(* Logix 5000 project; controller CLASE_1 Emulate 5570 rev 28.11; software revision 28.02; part 2 of 15 *)
(* tags used below, declared in another part *)
   Inp_PVSrcQ : SINT;   // Input Source and Quality (from Channel object, if available) (enum)
   Inp_PVBad : BOOL;   // 1=PV or I/O Comms Status Bad, 0=OK
   Inp_PVUncertain : BOOL;   // 1=PV Value Not Reliable, 0=OK
   Inp_Sim : BOOL;   // 1=Use simulated PV (Set_SimPV); 0=Use Input (Inp_PV)
   Cfg_UseChanSrcQ : BOOL;   // 1=Pass thru connected Channel's SrcQ value, 0=generate SrcQ
   Cfg_HiHiDB : REAL;   // High-High Status Deadband (EU)
   Cfg_HiDB : REAL;   // High Status Deadband (EU)
   Cfg_LoDB : REAL;   // Low Status Deadband (EU)
   Cfg_LoLoDB : REAL;   // Low-Low Status Deadband (EU)
   Cfg_FailDB : REAL;   // Out-of-Range (fail) High/Low Deadband (EU)
   PSet_Owner : DINT;   // Program Owner Request ID (non-zero) or Release (zero)
   PCmd_ClearCapt : BOOL;   // Program Command to Clear the captured min / max PV excursion values
   MCmd_SubstPV : BOOL;   // Maintenance Command to use Substitute PV (override input)
   MCmd_InpPV : BOOL;   // Maintenance Command to use Input PV (normal)
   OCmd_ResetAckAll : BOOL;   // Operator Command to Reset and Acknowledge all Alarms
   Val : REAL;   // Analog Value (after Substitute PV, if used)
   Val_InpPV : REAL;   // Analog Input Value (actual, before Substitute PV selection)
   SrcQ_IO : SINT;   // Source and Quality of primary I/O (enumeration)
   SrcQ : SINT;   // Source and Quality of primary Val/Sts (enumeration)
   Val_Fault : SINT;   // Device Fault Status 0=none, 20=Lo, 21=Hi, 24=LoLo, 25=HiHi, 32=Fail, 34=CfgErr
   Val_Owner : DINT;   // Current Object Owner ID (0=not owned)
   Sts_SubstPV : BOOL;   // 1=Using Substitute PV (Input being overridden)
   Err_Raw : BOOL;   // 1=Error in Config: Raw Input Scaling Min = Max
   Err_EU : BOOL;   // 1=Error in Config: Scaled EU Min = Max
   Err_Filt : BOOL;   // 1=Error in Config: PV filter params (RateTime, TC)
   Err_DB : BOOL;   // 1=Error in Config: a Status Deadband is < 0.0
   Err_Alarm : BOOL;   // 1=Error in Config: Alarm Min On Time, Shelf Time, Severity
   Sts_HiHi : ALIAS FOR HiHi.Inp;   // 1=Analog Input is above High-High limit
   Sts_Hi : ALIAS FOR Hi.Inp;   // 1=Analog Input is above High limit
   Sts_Lo : ALIAS FOR Lo.Inp;   // 1=Analog Input is below Low limit
   Sts_LoLo : ALIAS FOR LoLo.Inp;   // 1=Analog Input is below Low-Low limit
   Sts_Fail : ALIAS FOR Fail.Inp;   // 1=Analog Input is Out of Range or PV Bad
   Rdy_ResetAckAll : BOOL;   // 1=At least one Alarm requires Reset or Acknowledgement
   P_AIn : BOOL;   // Unique Parameter Name for auto - discovery
   LoLo : P_Alarm;   // Low-Low Alarm
   Lo : P_Alarm;   // Low Alarm
   Hi : P_Alarm;   // High Alarm
   HiHi : P_Alarm;   // High-High Alarm
   Mode : P_Mode;   // Analog Input Mode Selection
   Fail : P_Alarm;   // Analog Input Failure Alarm (bad quality or out of range)
   Wrk_Notify : SINT;   // Buffer for building Val_Notify
   Wrk_Fault : SINT;   // Buffer for building Val_Fault
   Wrk_SrcQ : SINT;   // Register for building Source / Quality enumeration
   Wrk_ValidONS : BOOL;   // Selected PV goes from Infinite or Not a Number to VALID
   Wrk_SelPVInfNaN : BOOL;   // Selected PV (Input or Substitute) is Infinite or NaN
   FailGate : P_Gate;   // Fail Alarm Gate / Delay Block
   Wrk_InpInfNaN : BOOL;   // Input is Infinite or Not a Number
   Wrk_InpFail : BOOL;   // Input Fail: out of range
(* P_AIn, continued *)

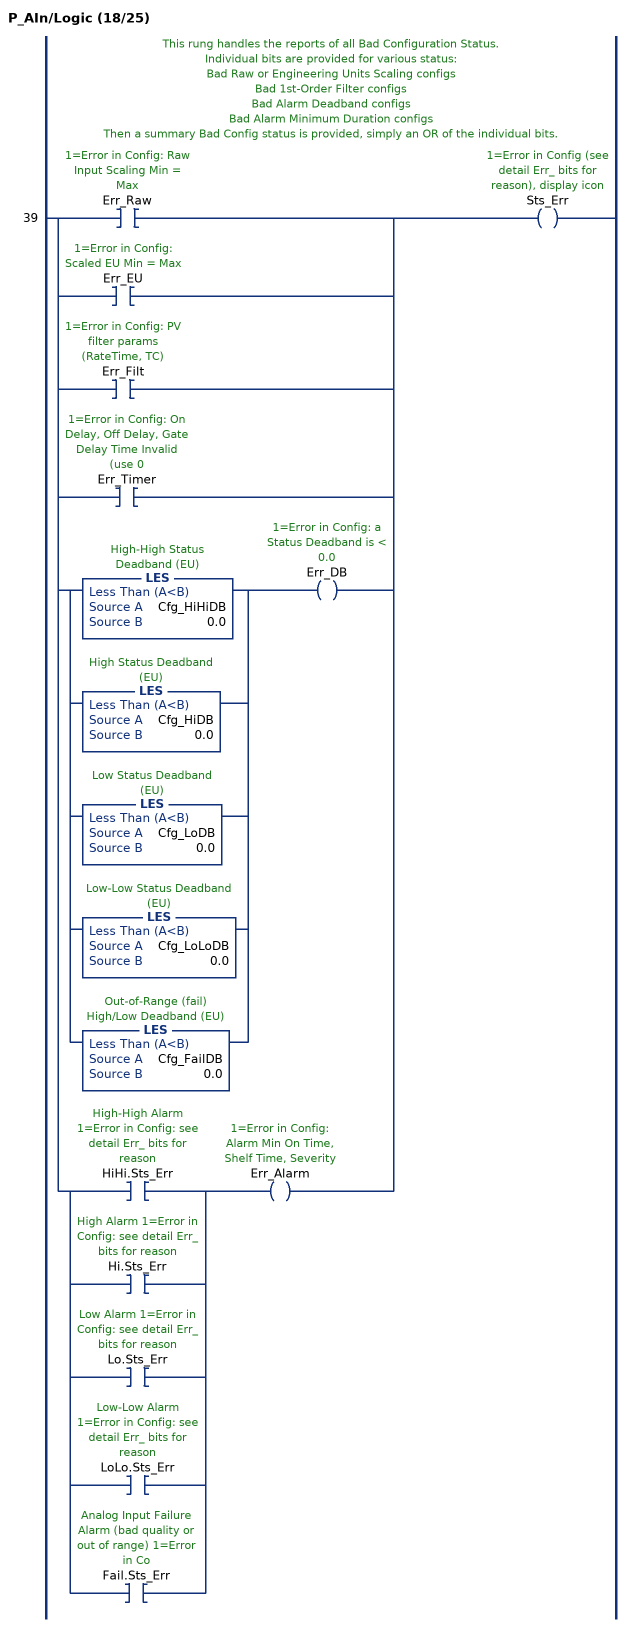
   // This rung handles the reports of all Bad Configuration Status.
   // Individual bits are provided for various status:
   // Bad Raw or Engineering Units Scaling configs
   // Bad 1st-Order Filter configs
   // Bad Alarm Deadband configs
   // Bad Alarm Minimum Duration configs
   // Then a summary Bad Config status is provided, simply an OR of the individual bits.
   39: [XIC(Err_Raw) ,XIC(Err_EU) ,XIC(Err_Filt) ,XIC(Err_Timer) ,[LES(Cfg_HiHiDB,0.0) ,LES(Cfg_HiDB,0.0) ,LES(Cfg_LoDB,0.0) ,LES(Cfg_LoLoDB,0.0) ,LES(Cfg_FailDB,0.0) ] OTE(Err_DB) ,[XIC(HiHi.Sts_Err) ,XIC(Hi.Sts_Err) ,XIC(Lo.Sts_Err) ,XIC(LoLo.Sts_Err) ,XIC(Fail.Sts_Err) ] OTE(Err_Alarm) ]OTE(Sts_Err);
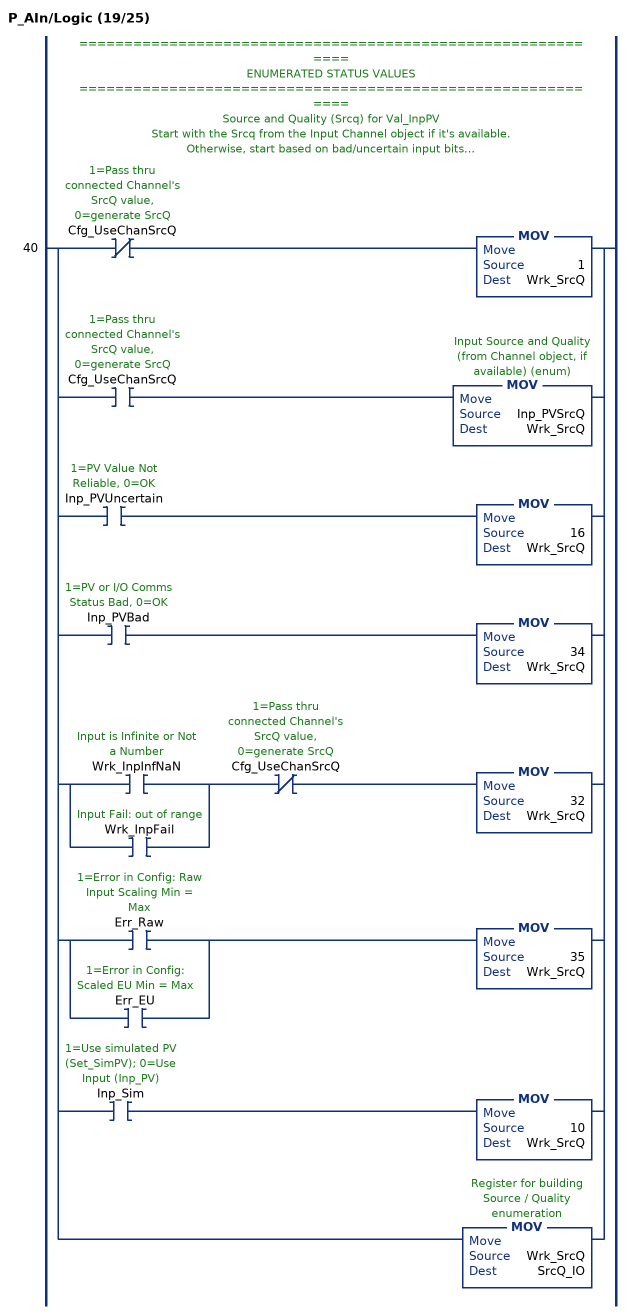
   // ============================================================
   // ENUMERATED STATUS VALUES
   // ============================================================
   // Source and Quality (Srcq) for Val_InpPV
   // Start with the Srcq from the Input Channel object if it's available.
   // Otherwise, start based on bad/uncertain input bits.
   // 0 = Good: live, confirmed good;   1 = Good: live, assumed good;
   // 2 = Good: no feedback, assumed good;   8 = Test: Simulated;   9 = Test: Loopback;
   // 10 = Test: Manually Entered;   16 = Uncertain: Live, off-spec;
   // 17 = Uncertain, Substituted at Device / Bus;   18 = Uncertain, Substituted at AOI;
   // 19 = Uncertain, using last known good;    20 = Uncertain, using replacement value;
   // 32 = Bad, Signal Failure;   33 = Bad, Channel Fault;
   // 34 = Bad, Module / Comms Fault;   35 = Bad, Invalid Configuration
   // #####  V3.1-00  2014-06-30:  Added rung for Source/Quality enumerations.  #####
   // #####  V3.5-02  2016-03-28:  Modified to add Cfg_UseChanSrcQ.  #####
   40: [XIO(Cfg_UseChanSrcQ) MOV(1,Wrk_SrcQ) ,XIC(Cfg_UseChanSrcQ) MOV(Inp_PVSrcQ,Wrk_SrcQ) ,XIC(Inp_PVUncertain) MOV(16,Wrk_SrcQ) ,XIC(Inp_PVBad) MOV(34,Wrk_SrcQ) ,[XIC(Wrk_InpInfNaN) ,XIC(Wrk_InpFail) ] XIO(Cfg_UseChanSrcQ) MOV(32,Wrk_SrcQ) ,[XIC(Err_Raw) ,XIC(Err_EU) ] MOV(35,Wrk_SrcQ) ,XIC(Inp_Sim) MOV(10,Wrk_SrcQ) ,MOV(Wrk_SrcQ,SrcQ_IO) ];
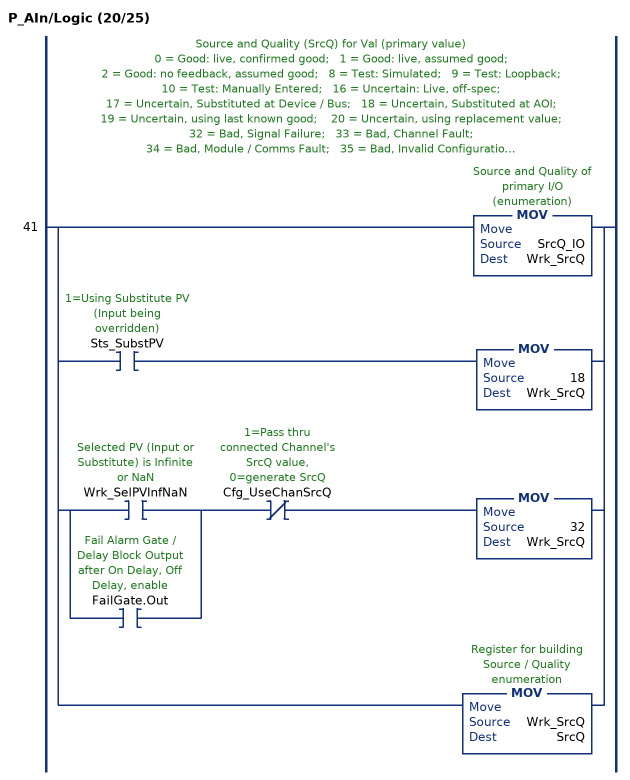
   // Source and Quality (SrcQ) for Val (primary value)
   // 0 = Good: live, confirmed good;   1 = Good: live, assumed good;
   // 2 = Good: no feedback, assumed good;   8 = Test: Simulated;   9 = Test: Loopback;
   // 10 = Test: Manually Entered;   16 = Uncertain: Live, off-spec;
   // 17 = Uncertain, Substituted at Device / Bus;   18 = Uncertain, Substituted at AOI;
   // 19 = Uncertain, using last known good;    20 = Uncertain, using replacement value;
   // 32 = Bad, Signal Failure;   33 = Bad, Channel Fault;
   // 34 = Bad, Module / Comms Fault;   35 = Bad, Invalid Configuration
   // #####  V3.1-00  2014-06-30:  Added rung for Source/Quality enumerations.  #####
   // #####  V3.5-02  2016-03-28:  Modified to add Cfg_UseChanSrcQ.  #####
   41: [MOV(SrcQ_IO,Wrk_SrcQ) ,XIC(Sts_SubstPV) MOV(18,Wrk_SrcQ) ,[XIC(Wrk_SelPVInfNaN) ,XIC(FailGate.Out) ] XIO(Cfg_UseChanSrcQ) MOV(32,Wrk_SrcQ) ,MOV(Wrk_SrcQ,SrcQ) ];
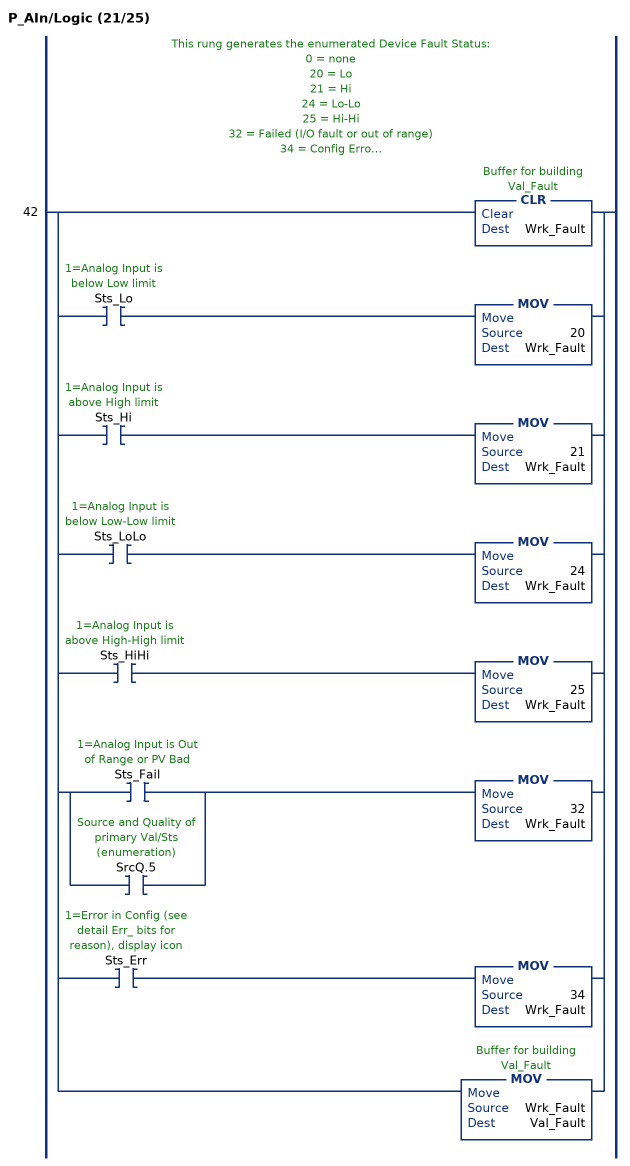
   // This rung generates the enumerated Device Fault Status:
   // 0 = none
   // 20 = Lo
   // 21 = Hi
   // 24 = Lo-Lo
   // 25 = Hi-Hi
   // 32 = Failed (I/O fault or out of range)
   // 34 = Config Error
   // #####  V3.1-05  2016-01-22:  Added check of SrcQ >= 32 for Val_Fault.  #####
   42: [CLR(Wrk_Fault) ,XIC(Sts_Lo) MOV(20,Wrk_Fault) ,XIC(Sts_Hi) MOV(21,Wrk_Fault) ,XIC(Sts_LoLo) MOV(24,Wrk_Fault) ,XIC(Sts_HiHi) MOV(25,Wrk_Fault) ,[XIC(Sts_Fail) ,XIC(SrcQ.5) ] MOV(32,Wrk_Fault) ,XIC(Sts_Err) MOV(34,Wrk_Fault) ,MOV(Wrk_Fault,Val_Fault) ];
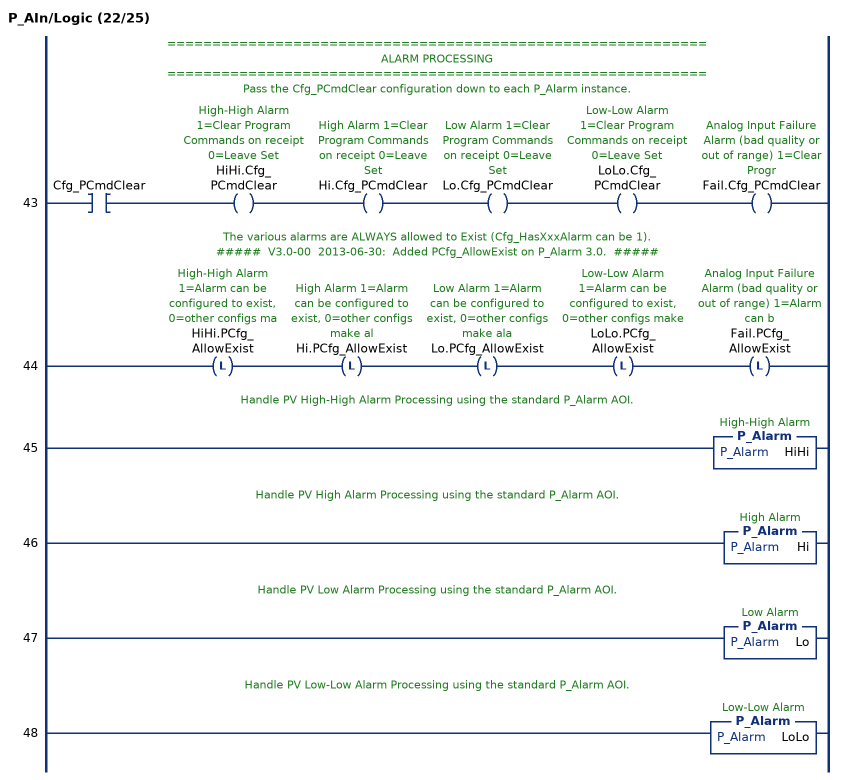
   // ============================================================
   // ALARM PROCESSING
   // ============================================================
   // Pass the Cfg_PCmdClear configuration down to each P_Alarm instance.
   43: XIC(Cfg_PCmdClear)OTE(HiHi.Cfg_PCmdClear)OTE(Hi.Cfg_PCmdClear)OTE(Lo.Cfg_PCmdClear)OTE(LoLo.Cfg_PCmdClear)OTE(Fail.Cfg_PCmdClear);
   // The various alarms are ALWAYS allowed to Exist (Cfg_HasXxxAlarm can be 1).
   // #####  V3.0-00  2013-06-30:  Added PCfg_AllowExist on P_Alarm 3.0.  #####
   44: OTL(HiHi.PCfg_AllowExist)OTL(Hi.PCfg_AllowExist)OTL(Lo.PCfg_AllowExist)OTL(LoLo.PCfg_AllowExist)OTL(Fail.PCfg_AllowExist);
   // Handle PV High-High Alarm Processing using the standard P_Alarm AOI.
   45: P_Alarm(HiHi);
   // Handle PV High Alarm Processing using the standard P_Alarm AOI.
   46: P_Alarm(Hi);
   // Handle PV Low Alarm Processing using the standard P_Alarm AOI.
   47: P_Alarm(Lo);
   // Handle PV Low-Low Alarm Processing using the standard P_Alarm AOI.
   48: P_Alarm(LoLo);
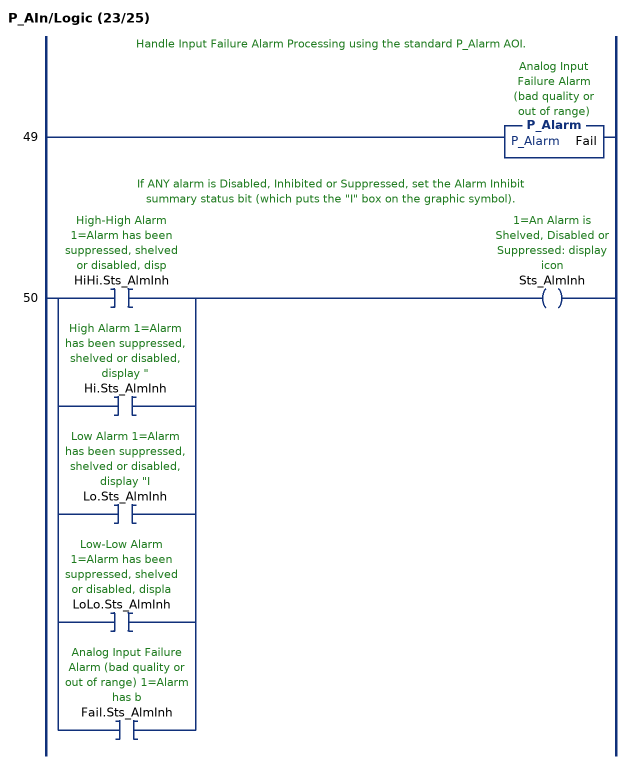
   // Handle Input Failure Alarm Processing using the standard P_Alarm AOI.
   49: P_Alarm(Fail);
   // If ANY alarm is Disabled, Inhibited or Suppressed, set the Alarm Inhibit
   // summary status bit (which puts the "I" box on the graphic symbol).
   50: [XIC(HiHi.Sts_AlmInh) ,XIC(Hi.Sts_AlmInh) ,XIC(Lo.Sts_AlmInh) ,XIC(LoLo.Sts_AlmInh) ,XIC(Fail.Sts_AlmInh) ]OTE(Sts_AlmInh);
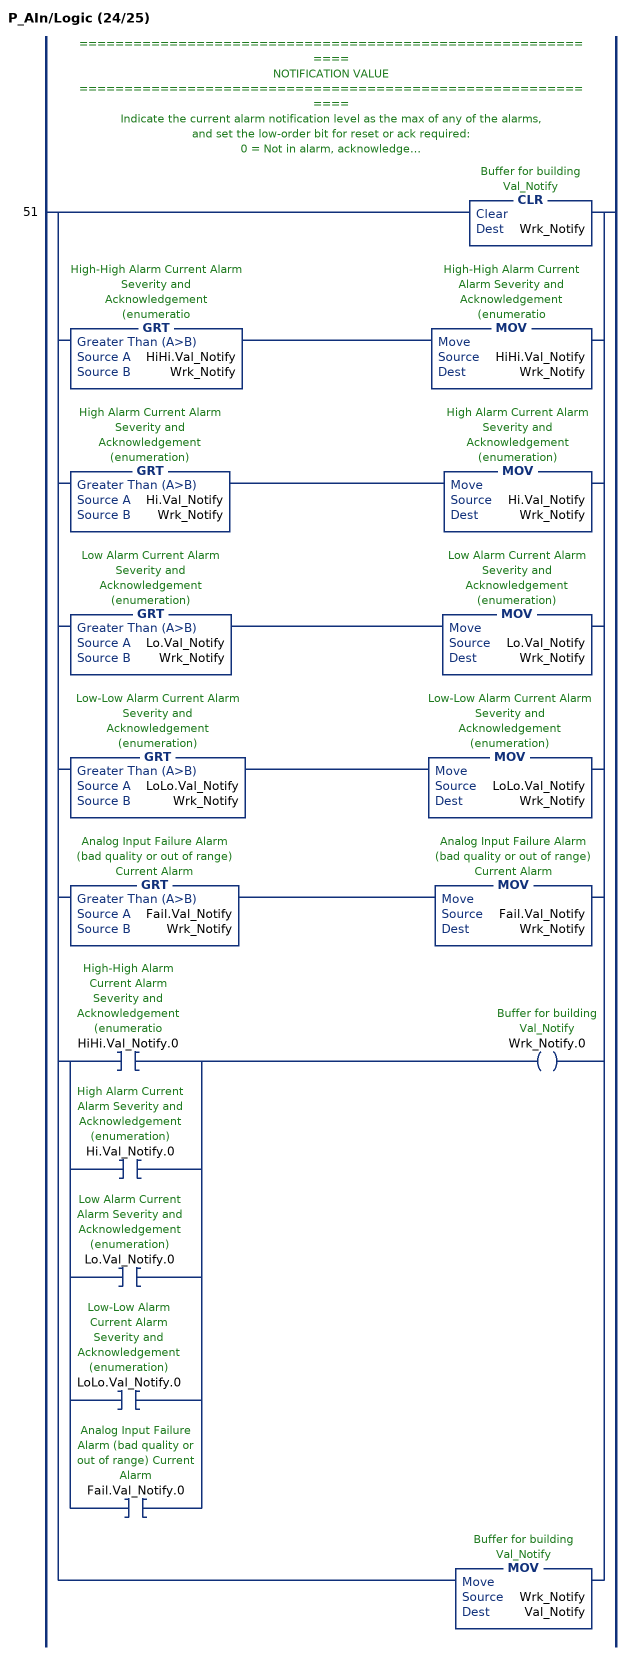
   // ============================================================
   // NOTIFICATION VALUE
   // ============================================================
   // Indicate the current alarm notification level as the max of any of the alarms,
   // and set the low-order bit for reset or ack required:
   // 0 = Not in alarm, acknowledged
   // 1 = Not in alarm, unacknowledged or reset required
   // 2 = Low severity alarm, acknowledged
   // 3 = Low severity alarm, unacknowledged
   // 4 = Medium severity alarm, acknowledged
   // 5 = Medium severity alarm, unacknowledged
   // 6 = High severity alarm, acknowledged
   // 7 = High severity alarm, unacknowledged
   // 8 = Urgent severity alarm, acknowledged
   // 9 = Urgent severity alarm, unacknowledged
   // #####  V3.1-00  2014-06-30:  Separated Reset Reqd functions from Val_Notify  #####
   51: [CLR(Wrk_Notify) ,GRT(HiHi.Val_Notify,Wrk_Notify) MOV(HiHi.Val_Notify,Wrk_Notify) ,GRT(Hi.Val_Notify,Wrk_Notify) MOV(Hi.Val_Notify,Wrk_Notify) ,GRT(Lo.Val_Notify,Wrk_Notify) MOV(Lo.Val_Notify,Wrk_Notify) ,GRT(LoLo.Val_Notify,Wrk_Notify) MOV(LoLo.Val_Notify,Wrk_Notify) ,GRT(Fail.Val_Notify,Wrk_Notify) MOV(Fail.Val_Notify,Wrk_Notify) ,[XIC(HiHi.Val_Notify.0) ,XIC(Hi.Val_Notify.0) ,XIC(Lo.Val_Notify.0) ,XIC(LoLo.Val_Notify.0) ,XIC(Fail.Val_Notify.0) ] OTE(Wrk_Notify.0) ,MOV(Wrk_Notify,Val_Notify) ];
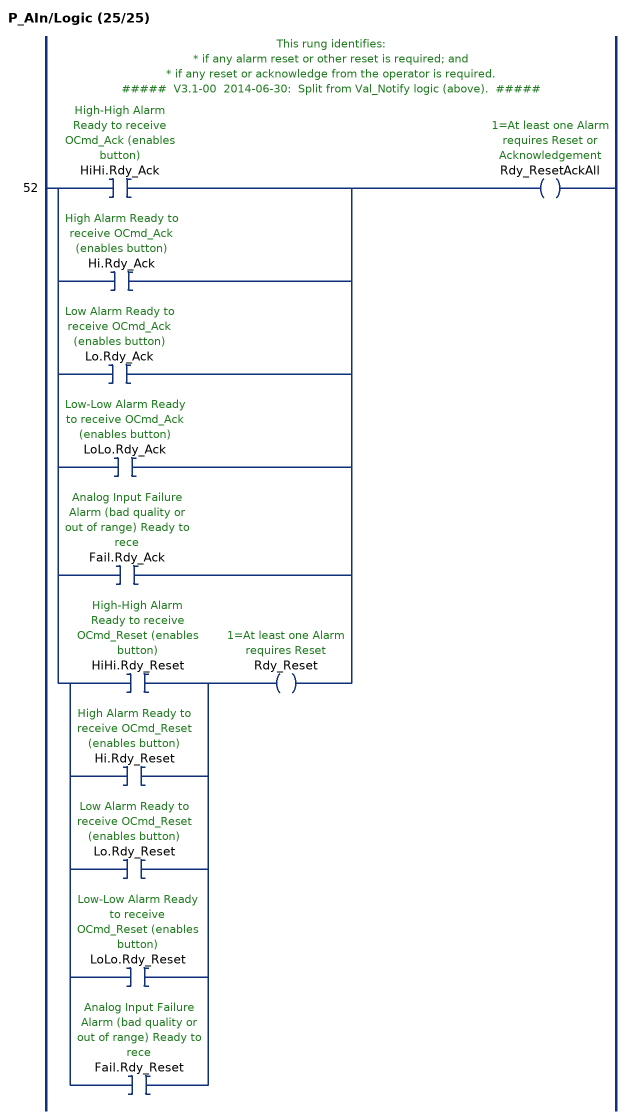
   // This rung identifies:
   // * if any alarm reset or other reset is required; and
   // * if any reset or acknowledge from the operator is required.
   // #####  V3.1-00  2014-06-30:  Split from Val_Notify logic (above).  #####
   52: [[XIC(HiHi.Rdy_Ack) ,XIC(Hi.Rdy_Ack) ,XIC(Lo.Rdy_Ack) ,XIC(LoLo.Rdy_Ack) ,XIC(Fail.Rdy_Ack) ] ,[XIC(HiHi.Rdy_Reset) ,XIC(Hi.Rdy_Reset) ,XIC(Lo.Rdy_Reset) ,XIC(LoLo.Rdy_Reset) ,XIC(Fail.Rdy_Reset) ] OTE(Rdy_Reset) ]OTE(Rdy_ResetAckAll);
END_ROUTINE

ROUTINE Prescan   (* ladder *)
// Clear Ownership. clear "lurking" Commands
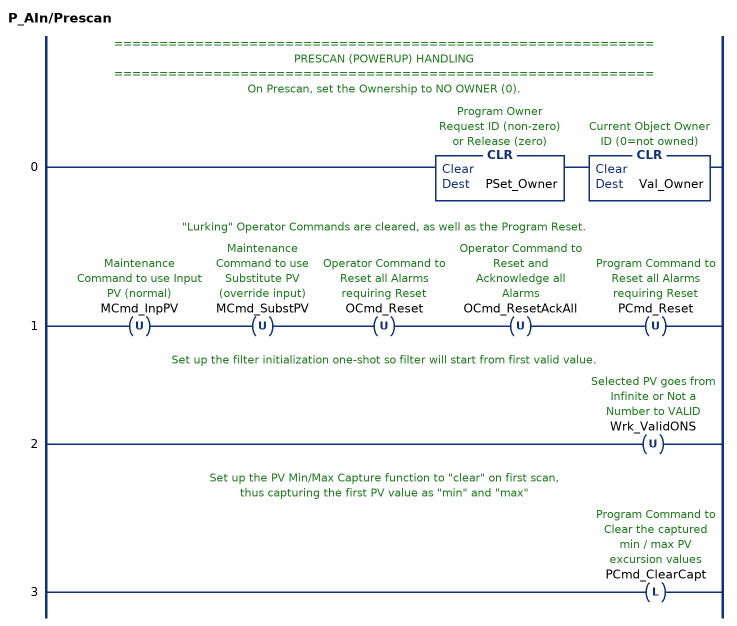
   // ============================================================
   // PRESCAN (POWERUP) HANDLING
   // ============================================================
   // On Prescan, set the Ownership to NO OWNER (0).
   0: CLR(PSet_Owner)CLR(Val_Owner);
   // "Lurking" Operator Commands are cleared, as well as the Program Reset.
   1: OTU(MCmd_InpPV)OTU(MCmd_SubstPV)OTU(OCmd_Reset)OTU(OCmd_ResetAckAll)OTU(PCmd_Reset);
   // Set up the filter initialization one-shot so filter will start from first valid value.
   2: OTU(Wrk_ValidONS);
   // Set up the PV Min/Max Capture function to "clear" on first scan,
   // thus capturing the first PV value as "min" and "max"
   3: OTL(PCmd_ClearCapt);
END_ROUTINE
END_ADD_ON_INSTRUCTION

ADD_ON_INSTRUCTION P_Alarm   (* revision 3.5 07Patch01 Release, vendor Rockwell Automation, ExecutePrescan, ExecuteEnableInFalse *)
// Alarm
// Revision note:
// See V3.5-xx Release Notes for details. Modified for FTView ME "chattering alarm" acknowledge timing.
// Help:
// Copyright © Rockwell Automation, Inc.  All Rights Reserved.
// This instruction monitors one input condition and provides one Alarm with:
//   * configurable latching (reset required) and acknowledgement requirement
//   * configurable alarm severity
//       1 to 250       = Low  (blue, typ. informational)
//       251 to 500   = Medium  (yelllow, typ. warning)
//       501 to 750   = High  (red, typ. process exception)
//       751 to 1000 = Urgent  (magenta, typ. equip. fault)
//   * configurable minimum ON time (e.g., to ensure it is seen by the HMI)
//   * commands to suppress/unsuppress (Prog), shelve/unshelve (Oper)
//         and disable/enable (Maint) the alarm.
//   * configurable amount of time shelved to automatically unshelve an alarm
//   * FTA&E support for suppressed, shelved and disabled states (V7.0)
//   * A Maintenance "Test" command, which triggers the alarm for the minimum
//      alarm time for testing purposes.
// NOTE regarding parameter naming:
//   FTAE names (same as ALMD instruction) are used instead
//   of the ANSI/ISA 18.2-2009 names, as follows:
//    "Disabled" is the equivalent of "Out of Service" in ISA 18.2.
//       (The Disabled state is owned by Maintenance.)
//    "Suppressed" is the equivalent of "Suppressed by Design" in
//       ISA 18.2. (The Suppressed state is owned by Program logic.)
//    "Shelved" is the same as in ISA 18.2.
//       (The Shelved state is owned by Operator, but may be cleared
//       by Program logic based on time, shift change, etc.)
// This instruction is usually nested within other instructions, with one instance
// used for each Alarm generated by the containing instruction.  It may also be
// used as a standalone instruction for Alarm conditions generated by custom logic.
// FTAE Alarm Setup:
//   (object).(alarm).Com_AE.0:  Alarm to FTAE
//     .Com_AE.1:   Ack to/from FTAE
//     .Com_AE.3:   Shelved from FTAE Status
//     .Com_AE.4:   Shelve/Reshelve to FTAE Control (auto reset)
//     .Com_AE.5:   Unshelve to FTAE Control (auto reset)
//     .Com_AE.6:   Suppressed from FTAE Status
//     .Com_AE.7:   Suppress to FTAE Control (auto reset)
//     .Com_AE.8:   Unsuppress to FTAE Control (auto reset)
//     .Com_AE.9:   Disabled from FTAE Status
//     .Com_AE.10: Disable to FTAE Control (auto reset)
//     .Com_AE.11: Enable to FTAE Control (auto reset)
//    all other bits unused
//     .Cfg_MaxShelfT is also used in FTAE config.
//     .Cfg_Severity is used in FTAE for FTView 8.x.
VAR_INPUT
   Inp : BOOL := 1; {visible}   // Alarm Condition Input 1=Alarm
   Inp_Reset : BOOL; {visible}   // 1=Reset Alarm requiring reset
   Cfg_Exists : BOOL := 1;   // 1=Alarm configured to exist, 0=Does not exist, don't scan
   Cfg_ResetReqd : BOOL;   // 1=Latched Alarm, a Reset is required to clear this Alarm
   Cfg_AckReqd : BOOL := 1;   // 1=Acknowledge required for this Alarm
   Cfg_AllowShelve : BOOL := 1;   // 1=Allow Operator to Shelve this Alarm
   Cfg_AllowDisable : BOOL := 1;   // 1=Allow Maintenance to Disable this Alarm
   Cfg_PCmdClear : BOOL := 1;   // 1=Clear Program Commands on receipt 0=Leave Set
   Cfg_Severity : INT := 750;   // Alarm Severity: 1..250=Low, 251..500=Medium, 501..750=High, 751..1000=Urgent
   Cfg_AlmMinOnT : DINT := 5;   // Minimum time Alm output stays on (sec)
   Cfg_MaxShelfT : INT := 480;   // Auto unshelve after shelved this long (1..32767 minutes)
   PCfg_AllowExist : BOOL := 1;   // 1=Alarm can be configured to exist, 0=other configs make alarm meaningless
   PCmd_Reset : BOOL;   // Program Command to Reset latched alarm
   PCmd_Ack : BOOL;   // Program Command to Acknowledge alarm
   PCmd_Suppress : BOOL;   // Program Command to Suppress by Design (inhibits new alarm)
   PCmd_Unsuppress : BOOL;   // Program Command to Unsuppress (allows new alarm)
   PCmd_Unshelve : BOOL;   // Program Command to Unshelve (e.g., on shift change)
   OCmd_Reset : BOOL;   // Operator Command to Reset latched alarm
   OCmd_Ack : BOOL;   // Operator Command to Acknowledge alarm
   OCmd_Shelve : BOOL;   // Operator Command to Shelve Alarm (inhibits new alarm)
   OCmd_Unshelve : BOOL;   // Operator Command to Unshelve alarm (allows new alarm)
   MCmd_Disable : BOOL;   // Maintenance Command to Disable alarm (inhibits new alarm)
   MCmd_Enable : BOOL;   // Maintenance Command to Enable alarm (allows new alarm)
   MCmd_Test : BOOL;   // Maintenance Command to Test alarm (issued for minimum alarm time)
END_VAR
VAR_OUTPUT
   Val_Notify : SINT; {access Read Only}   // Current Alarm Severity and Acknowledgement (enumeration)
   Val_MinToUnshelve : DINT; {access Read Only, visible}   // Number of minutes until this alarm unshelves itself (mmm:ss)
   Val_SecToUnshelve : DINT; {access Read Only, visible}   // Number of Seconds until this alarm unshelves itself (mmm:ss)
   Alm : ALIAS FOR Com_AE.0; {visible}   // Alarm output 1=In Alarm
   Ack : ALIAS FOR Com_AE.1; {visible}   // Alarm acknowledged status: 1=Ack rcvd
   Shelved : ALIAS FOR Com_AE.3; {visible}   // 1=Alarm has been Shelved by Operator (inhibits new alarm)
   Suppressed : ALIAS FOR Com_AE.6; {visible}   // 1=Alarm has been Suppressed by Program (inhibits new alarm)
   Disabled : ALIAS FOR Com_AE.9; {visible}   // 1=Alarm has been Disabled by Maintanance (inhibits new alarm)
   Sts_AlmInh : BOOL; {access Read Only}   // 1=Alarm has been suppressed, shelved or disabled, display "I" icon
   Sts_Err : BOOL; {access Read Only}   // 1=Error in Config: see detail Err_ bits for reason
   Err_Timer : BOOL; {access Read Only}   // 1=Error in Config: Alarm Min On Time, Shelf Time (use 0 to 2147483)
   Err_Severity : BOOL; {access Read Only}   // 1=Error in Config: Invalid Severity (use 1 to 4)
   Rdy_Reset : BOOL; {access Read Only}   // Ready to receive OCmd_Reset (enables button)
   Rdy_Ack : BOOL; {access Read Only}   // Ready to receive OCmd_Ack (enables button)
   Rdy_Shelve : BOOL; {access Read Only}   // Ready to receive OCmd_Shelve (enables button)
   Rdy_Unshelve : BOOL; {access Read Only}   // Ready to receive OCmd_Unshelve (enables button)
   Rdy_Disable : BOOL; {access Read Only}   // Ready to receive MCmd_Disable (enables button)
   Rdy_Enable : BOOL; {access Read Only}   // Ready to receive MCmd_Enable (enables button)
   Rdy_Test : BOOL; {access Read Only}   // Ready to receive MCmd_Test (enables button)
   P_Alarm : BOOL;   // Unique Parameter Name for auto - discovery
END_VAR
VAR
   Wrk_Alm : BOOL; {access None}   // Internal Alarm Status
   Wrk_Suppressed : BOOL; {access None}   // Internal Alarm Suppressed Status
   Wrk_AlmMinOnT : TIMER := (PRE := 5000); {access None}   // Alarm output minimum ON time to be seen by alarm server
   Wrk_AutoAckT : TIMER := (PRE := 5000); {access None}   // Time to clear Ack bit when Ack not required
   Wrk_ShelfT : TIMER; {access Read Only}   // Time to auto Unshelve a Shelved Alarm
   Inf_Tab : SINT;   // Tab to display (FTView ME)
   Com_AE : INT := 2#0000_0000_0000_0010;   // Communication with HMI / Alarm/Event Server (see bit descriptions)
        .0   // Alarm to AE
        .1   // Acked from AE Status, Ack to AE Control
        .10   // Disable to AE Control
        .11   // Enable to AE Control
        .12   // (not used)
        .13   // (not used)
        .14   // (not used)
        .15   // (not used)
        .2   // (not used)
        .3   // Shelved from AE Status
        .4   // Shelve to AE Control
        .5   // Unshelve to AE Control
        .6   // Suppressed from AE Status
        .7   // Suppress to AE Control
        .8   // Unsuppress to AE Control
        .9   // Disabled from AE Status
   Cfg_Tag : STRING_20 := 'P_Alarm';   // Alarm Tag Text (e.g., "LAHH-101")
   Cfg_Cond : STRING_20 := 'Alarm Condition';   // Alarm Condition Text (e.g., "High-High PV")
   Wrk_SecToUnshelve : DINT; {access None}   // Number of seconds until this alarm unshelves itself
   Inf_Lib : STRING_12 := 'RA-BAS'; {access Read Only}   // Display Library for Faceplate call-up
   Inf_Type : STRING_16 := 'P_Alarm'; {access Read Only}   // Must contain AOI name, used for HMI and Information S/W
END_VAR

ROUTINE EnableInFalse   (* ladder *)
// Perform Alarm processing, but Invert Alarm Input ("Inp") for use on LD rung (EnableIn False)
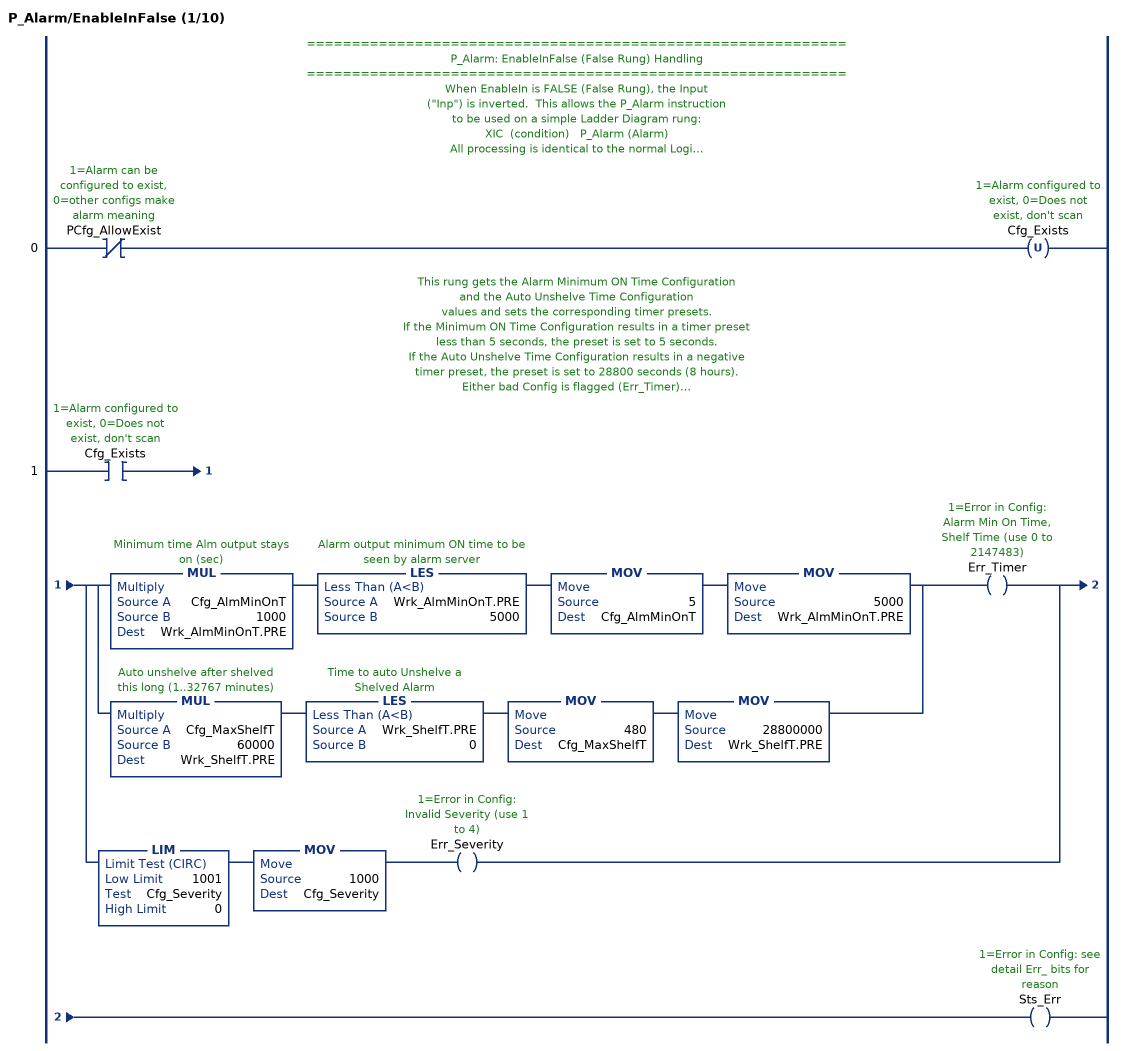
   // ============================================================
   // P_Alarm: EnableInFalse (False Rung) Handling
   // ============================================================
   // When EnableIn is FALSE (False Rung), the Input
   // ("Inp") is inverted.  This allows the P_Alarm instruction
   // to be used on a simple Ladder Diagram rung:
   // XIC  (condition)   P_Alarm (Alarm)
   // All processing is identical to the normal Logic
   // routine, except references to Inp are inverted!
   // ============================================================
   // CONFIGURATION
   // ============================================================
   // In the object containing this alarm, other configuration (such as not having
   // any limit switches) may make this particular alarm meaningless.
   // The Program Configuration "Allow Exist" is used to hide this alarm
   // on the object's faceplate and other graphics, and forces the Cfg_Exist to 0.
   // #####  V3.0-00  2013-06-30:  Added PCfg_AllowExist.  #####
   0: XIO(PCfg_AllowExist)OTU(Cfg_Exists);
   // This rung gets the Alarm Minimum ON Time Configuration
   // and the Auto Unshelve Time Configuration
   // values and sets the corresponding timer presets.
   // If the Minimum ON Time Configuration results in a timer preset
   // less than 5 seconds, the preset is set to 5 seconds.
   // If the Auto Unshelve Time Configuration results in a negative
   // timer preset, the preset is set to 28800 seconds (8 hours).
   // Either bad Config is flagged (Err_Timer).
   // Bad Config is also flagged if the Cfg_Severity is out of range (valid = 1..1000) (Err_Severity).
   // #####  V3.0-00  2013-06-30:  Changed Program Inhibit to Suppress, Operator Suppress to Shelve.  #####
   // #####  Added Shelf Timer config check; if Severity out of range, make it "Fault".  #####
   // #####  V3.0-02  2013-10-30:  Changed Cfg_MaxShelfT check to LEQ 0.  (INT 1 to 32767 is valid.)  #####
   // #####  V3.1-05, V3.5-00  2015-07-31:  Fixed operation of Cfg_MaxShelfT = 0, Cfg_AlmMinOnT, rung comment.  #####
   1: XIC(Cfg_Exists)[[MUL(Cfg_AlmMinOnT,1000,Wrk_AlmMinOnT.PRE) LES(Wrk_AlmMinOnT.PRE,5000) MOV(5,Cfg_AlmMinOnT) MOV(5000,Wrk_AlmMinOnT.PRE) ,MUL(Cfg_MaxShelfT,60000,Wrk_ShelfT.PRE) LES(Wrk_ShelfT.PRE,0) MOV(480,Cfg_MaxShelfT) MOV(28800000,Wrk_ShelfT.PRE) ] OTE(Err_Timer) ,LIM(1001,Cfg_Severity,0) MOV(1000,Cfg_Severity) OTE(Err_Severity) ]OTE(Sts_Err);
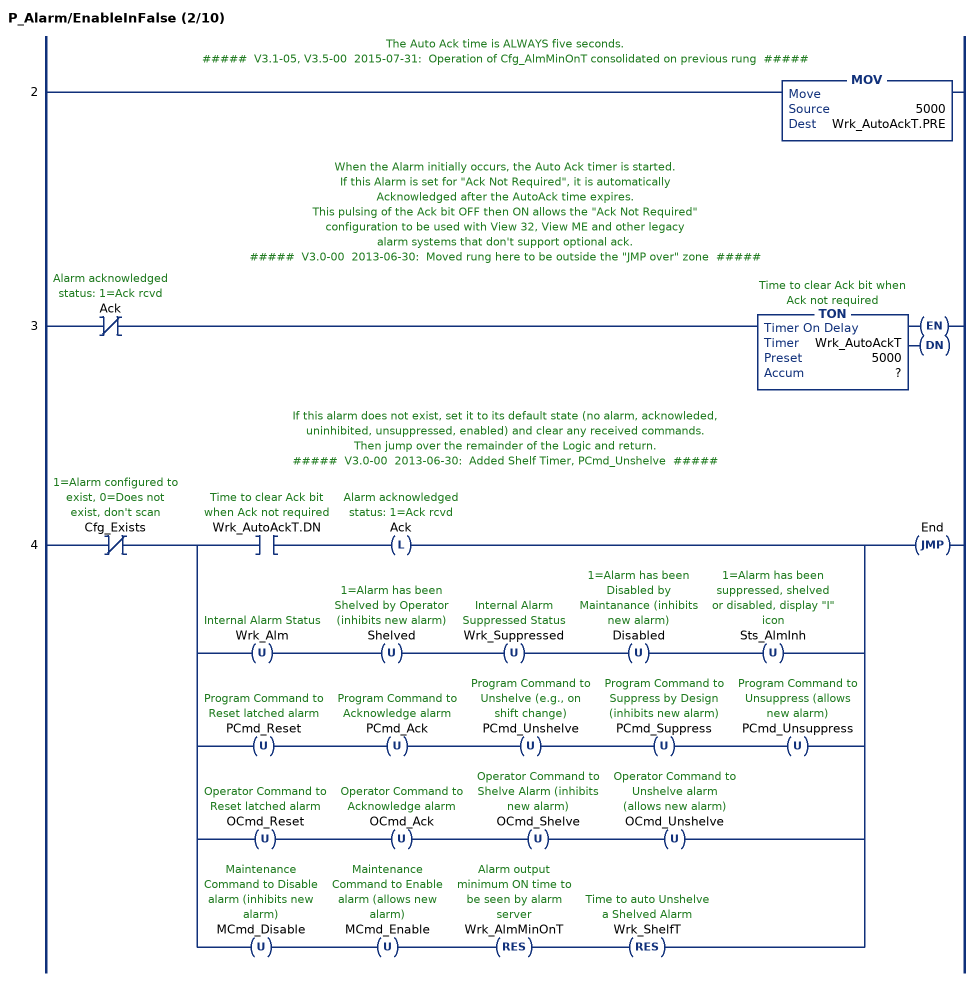
   // The Auto Ack time is ALWAYS five seconds.
   // #####  V3.1-05, V3.5-00  2015-07-31:  Operation of Cfg_AlmMinOnT consolidated on previous rung  #####
   2: MOV(5000,Wrk_AutoAckT.PRE);
   // When the Alarm initially occurs, the Auto Ack timer is started.
   // If this Alarm is set for "Ack Not Required", it is automatically
   // Acknowledged after the AutoAck time expires.
   // This pulsing of the Ack bit OFF then ON allows the "Ack Not Required"
   // configuration to be used with View 32, View ME and other legacy
   // alarm systems that don't support optional ack.
   // #####  V3.0-00  2013-06-30:  Moved rung here to be outside the "JMP over" zone  #####
   3: XIO(Ack)TON(Wrk_AutoAckT,?,?);
   // If this alarm does not exist, set it to its default state (no alarm, acknowleded,
   // uninhibited, unsuppressed, enabled) and clear any received commands.
   // Then jump over the remainder of the Logic and return.
   // #####  V3.0-00  2013-06-30:  Added Shelf Timer, PCmd_Unshelve  #####
   4: XIO(Cfg_Exists)[XIC(Wrk_AutoAckT.DN) OTL(Ack) ,OTU(Wrk_Alm) OTU(Shelved) OTU(Wrk_Suppressed) OTU(Disabled) OTU(Sts_AlmInh) ,OTU(PCmd_Reset) OTU(PCmd_Ack) OTU(PCmd_Unshelve) OTU(PCmd_Suppress) OTU(PCmd_Unsuppress) ,OTU(OCmd_Reset) OTU(OCmd_Ack) OTU(OCmd_Shelve) OTU(OCmd_Unshelve) ,OTU(MCmd_Disable) OTU(MCmd_Enable) RES(Wrk_AlmMinOnT) RES(Wrk_ShelfT) ]JMP(End);
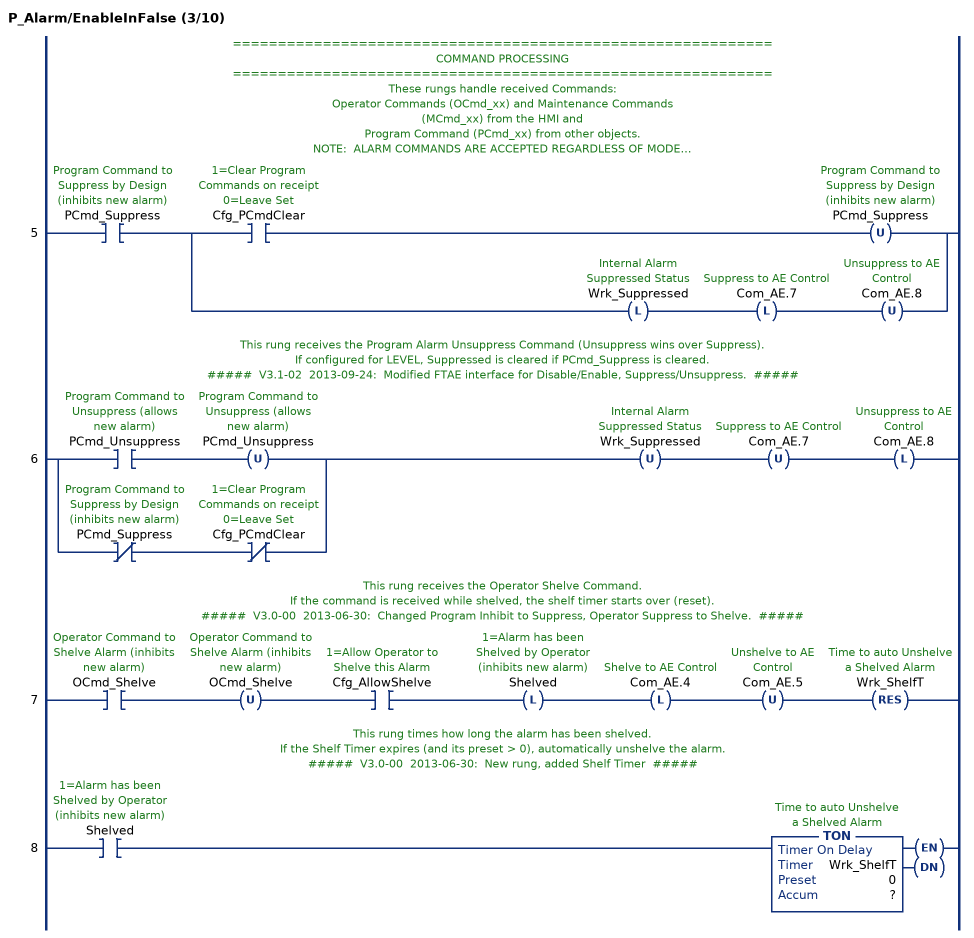
   // ============================================================
   // COMMAND PROCESSING
   // ============================================================
   // These rungs handle received Commands:
   // Operator Commands (OCmd_xx) and Maintenance Commands
   // (MCmd_xx) from the HMI and
   // Program Command (PCmd_xx) from other objects.
   // NOTE:  ALARM COMMANDS ARE ACCEPTED REGARDLESS OF MODE.
   // This rung receives the Program Alarm Inhibit Command.
   // If configured for EDGE, the Command is cleared.
   // #####  V3.1-02  2013-09-24:  Modified FTAE interface for Disable/Enable, Suppress/Unsuppress.  #####
   5: XIC(PCmd_Suppress)[XIC(Cfg_PCmdClear) OTU(PCmd_Suppress) ,OTL(Wrk_Suppressed) OTL(Com_AE.7) OTU(Com_AE.8) ];
   // This rung receives the Program Alarm Unsuppress Command (Unsuppress wins over Suppress).
   // If configured for LEVEL, Suppressed is cleared if PCmd_Suppress is cleared.
   // #####  V3.1-02  2013-09-24:  Modified FTAE interface for Disable/Enable, Suppress/Unsuppress.  #####
   6: [XIC(PCmd_Unsuppress) OTU(PCmd_Unsuppress) ,XIO(PCmd_Suppress) XIO(Cfg_PCmdClear) ]OTU(Wrk_Suppressed)OTU(Com_AE.7)OTL(Com_AE.8);
   // This rung receives the Operator Shelve Command.
   // If the command is received while shelved, the shelf timer starts over (reset).
   // #####  V3.0-00  2013-06-30:  Changed Program Inhibit to Suppress, Operator Suppress to Shelve.  #####
   7: XIC(OCmd_Shelve)OTU(OCmd_Shelve)XIC(Cfg_AllowShelve)OTL(Shelved)OTL(Com_AE.4)OTU(Com_AE.5)RES(Wrk_ShelfT);
   // This rung times how long the alarm has been shelved.
   // If the Shelf Timer expires (and its preset > 0), automatically unshelve the alarm.
   // #####  V3.0-00  2013-06-30:  New rung, added Shelf Timer  #####
   8: XIC(Shelved)TON(Wrk_ShelfT,?,?);
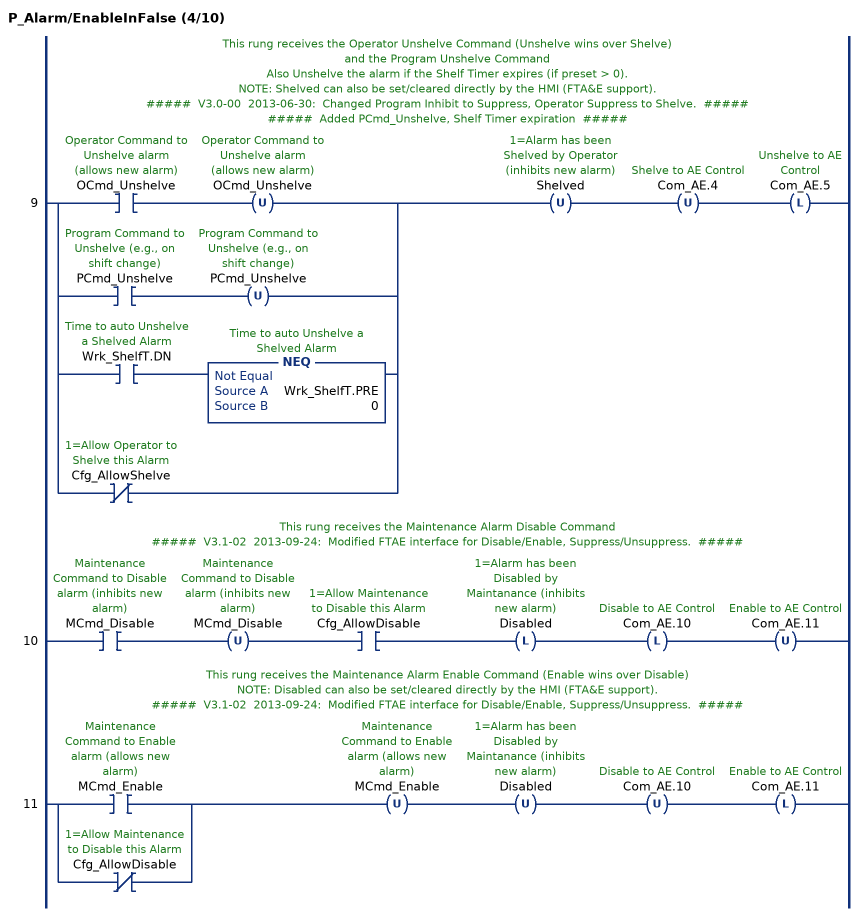
   // This rung receives the Operator Unshelve Command (Unshelve wins over Shelve)
   // and the Program Unshelve Command
   // Also Unshelve the alarm if the Shelf Timer expires (if preset > 0).
   // NOTE: Shelved can also be set/cleared directly by the HMI (FTA&E support).
   // #####  V3.0-00  2013-06-30:  Changed Program Inhibit to Suppress, Operator Suppress to Shelve.  #####
   // #####  Added PCmd_Unshelve, Shelf Timer expiration  #####
   9: [XIC(OCmd_Unshelve) OTU(OCmd_Unshelve) ,XIC(PCmd_Unshelve) OTU(PCmd_Unshelve) ,XIC(Wrk_ShelfT.DN) NEQ(Wrk_ShelfT.PRE,0) ,XIO(Cfg_AllowShelve) ]OTU(Shelved)OTU(Com_AE.4)OTL(Com_AE.5);
   // This rung receives the Maintenance Alarm Disable Command
   // #####  V3.1-02  2013-09-24:  Modified FTAE interface for Disable/Enable, Suppress/Unsuppress.  #####
   10: XIC(MCmd_Disable)OTU(MCmd_Disable)XIC(Cfg_AllowDisable)OTL(Disabled)OTL(Com_AE.10)OTU(Com_AE.11);
   // This rung receives the Maintenance Alarm Enable Command (Enable wins over Disable)
   // NOTE: Disabled can also be set/cleared directly by the HMI (FTA&E support).
   // #####  V3.1-02  2013-09-24:  Modified FTAE interface for Disable/Enable, Suppress/Unsuppress.  #####
   11: [XIC(MCmd_Enable) ,XIO(Cfg_AllowDisable) ]OTU(MCmd_Enable)OTU(Disabled)OTU(Com_AE.10)OTL(Com_AE.11);
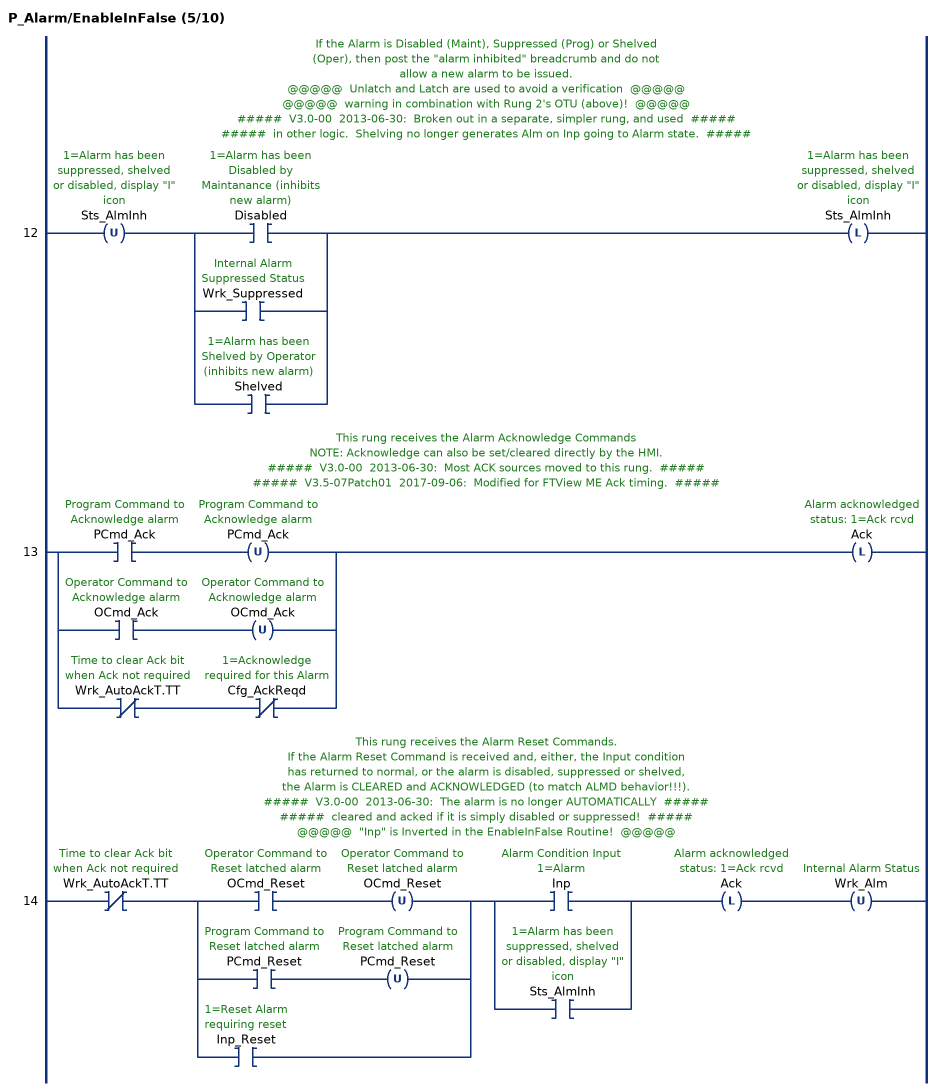
   // If the Alarm is Disabled (Maint), Suppressed (Prog) or Shelved
   // (Oper), then post the "alarm inhibited" breadcrumb and do not
   // allow a new alarm to be issued.
   // @@@@@  Unlatch and Latch are used to avoid a verification  @@@@@
   // @@@@@  warning in combination with Rung 2's OTU (above)!  @@@@@
   // #####  V3.0-00  2013-06-30:  Broken out in a separate, simpler rung, and used  #####
   // #####  in other logic.  Shelving no longer generates Alm on Inp going to Alarm state.  #####
   12: OTU(Sts_AlmInh)[XIC(Disabled) ,XIC(Wrk_Suppressed) ,XIC(Shelved) ]OTL(Sts_AlmInh);
   // This rung receives the Alarm Acknowledge Commands
   // NOTE: Acknowledge can also be set/cleared directly by the HMI.
   // #####  V3.0-00  2013-06-30:  Most ACK sources moved to this rung.  #####
   // #####  V3.5-07Patch01  2017-09-06:  Modified for FTView ME Ack timing.  #####
   13: [XIC(PCmd_Ack) OTU(PCmd_Ack) ,XIC(OCmd_Ack) OTU(OCmd_Ack) ,XIO(Wrk_AutoAckT.TT) XIO(Cfg_AckReqd) ]OTL(Ack);
   // This rung receives the Alarm Reset Commands.
   // If the Alarm Reset Command is received and, either, the Input condition
   // has returned to normal, or the alarm is disabled, suppressed or shelved,
   // the Alarm is CLEARED and ACKNOWLEDGED (to match ALMD behavior!!!).
   // #####  V3.0-00  2013-06-30:  The alarm is no longer AUTOMATICALLY  #####
   // #####  cleared and acked if it is simply disabled or suppressed!  #####
   // @@@@@  "Inp" is Inverted in the EnableInFalse Routine!  @@@@@
   14: XIO(Wrk_AutoAckT.TT)[XIC(OCmd_Reset) OTU(OCmd_Reset) ,XIC(PCmd_Reset) OTU(PCmd_Reset) ,XIC(Inp_Reset) ][XIC(Inp) ,XIC(Sts_AlmInh) ]OTL(Ack)OTU(Wrk_Alm);
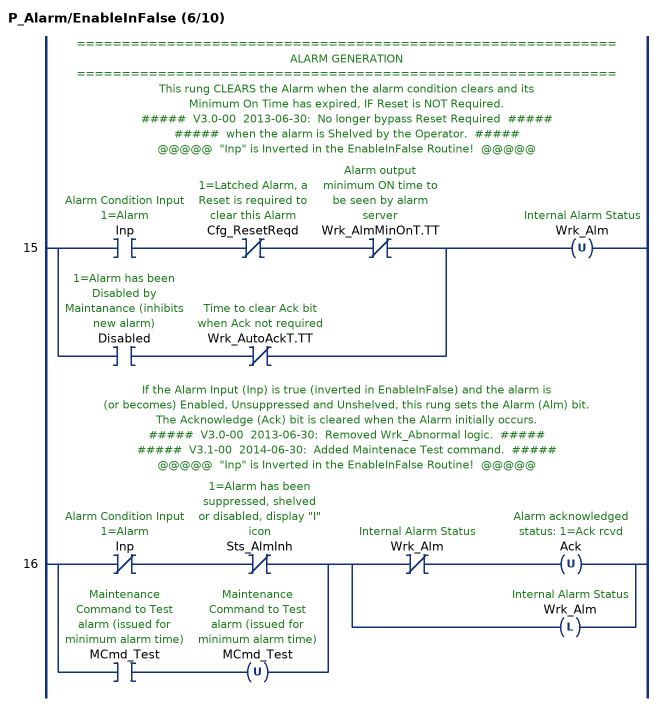
   // ============================================================
   // ALARM GENERATION
   // ============================================================
   // This rung CLEARS the Alarm when the alarm condition clears and its
   // Minimum On Time has expired, IF Reset is NOT Required.
   // #####  V3.0-00  2013-06-30:  No longer bypass Reset Required  #####
   // #####  when the alarm is Shelved by the Operator.  #####
   // @@@@@  "Inp" is Inverted in the EnableInFalse Routine!  @@@@@
   15: [XIC(Inp) XIO(Cfg_ResetReqd) XIO(Wrk_AlmMinOnT.TT) ,XIC(Disabled) XIO(Wrk_AutoAckT.TT) ]OTU(Wrk_Alm);
   // If the Alarm Input (Inp) is true (inverted in EnableInFalse) and the alarm is
   // (or becomes) Enabled, Unsuppressed and Unshelved, this rung sets the Alarm (Alm) bit.
   // The Acknowledge (Ack) bit is cleared when the Alarm initially occurs.
   // #####  V3.0-00  2013-06-30:  Removed Wrk_Abnormal logic.  #####
   // #####  V3.1-00  2014-06-30:  Added Maintenace Test command.  #####
   // @@@@@  "Inp" is Inverted in the EnableInFalse Routine!  @@@@@
   16: [XIO(Inp) XIO(Sts_AlmInh) ,XIC(MCmd_Test) OTU(MCmd_Test) ][XIO(Wrk_Alm) OTU(Ack) ,OTL(Wrk_Alm) ];
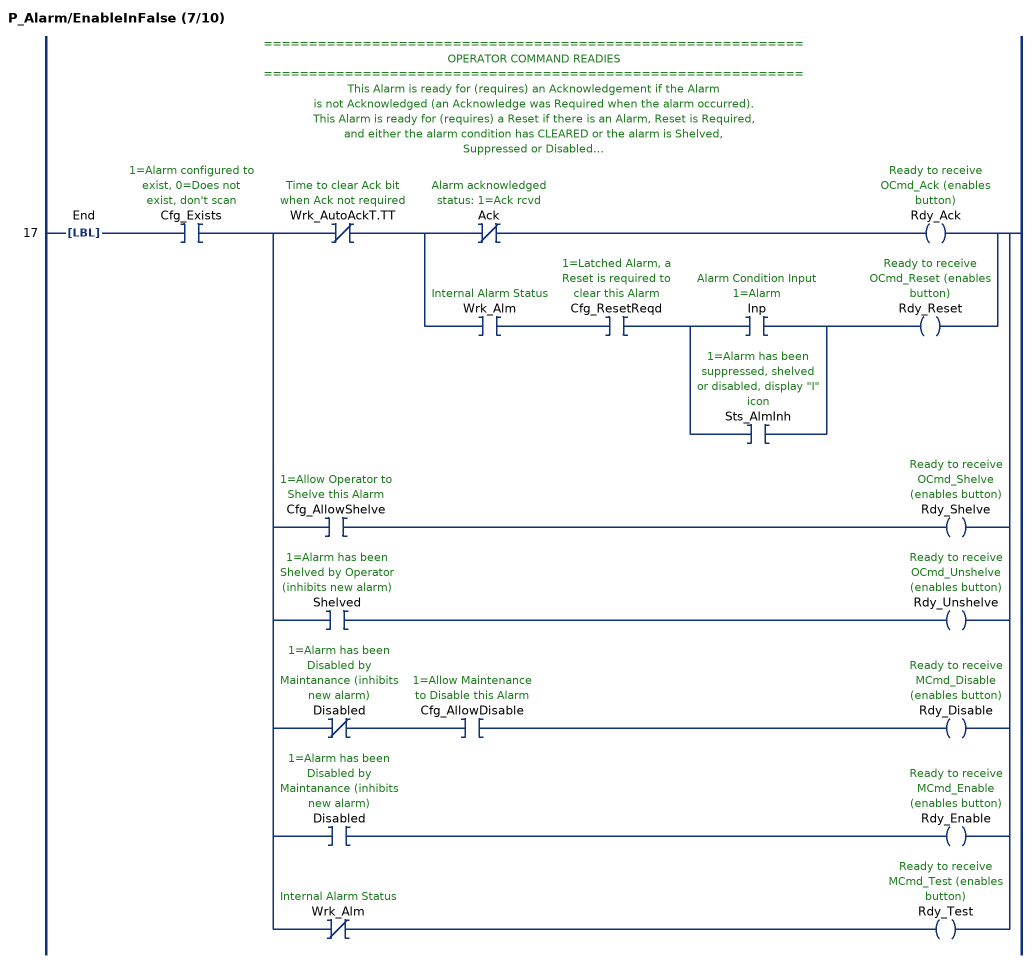
   // ============================================================
   // OPERATOR COMMAND READIES
   // ============================================================
   // This Alarm is ready for (requires) an Acknowledgement if the Alarm
   // is not Acknowledged (an Acknowledge was Required when the alarm occurred).
   // This Alarm is ready for (requires) a Reset if there is an Alarm, Reset is Required,
   // and either the alarm condition has CLEARED or the alarm is Shelved,
   // Suppressed or Disabled.
   // .
   // If the Alarm is NOT Shelved, it is ready for Shelve.
   // If the Alarm IS Shelved, it is ready for Unshelve.
   // If the Alarm is NOT Disabled, it is ready for Disable.
   // If the Alarm IS Disabled, it is ready for Enable.
   // NOTE: This rung appears before the Values/Status rung because the Rdy_Reset
   // condition is used to eliminate redundant logic in the rung below for Val_Notify.0.
   // #####  V3.0-00  2013-06-30:  Added sub-branch with Sts_AlmInh  #####
   // #####  V3.1-00  2014-06-30:  Added Maintenace Test command.  #####
   // @@@@@  "Inp" is Inverted in the EnableInFalse Routine!  @@@@@
   17: LBL(End)XIC(Cfg_Exists)[XIO(Wrk_AutoAckT.TT) [XIO(Ack) OTE(Rdy_Ack) ,XIC(Wrk_Alm) XIC(Cfg_ResetReqd) [XIC(Inp) ,XIC(Sts_AlmInh) ] OTE(Rdy_Reset) ] ,XIC(Cfg_AllowShelve) OTE(Rdy_Shelve) ,XIC(Shelved) OTE(Rdy_Unshelve) ,XIO(Disabled) XIC(Cfg_AllowDisable) OTE(Rdy_Disable) ,XIC(Disabled) OTE(Rdy_Enable) ,XIO(Wrk_Alm) OTE(Rdy_Test) ];
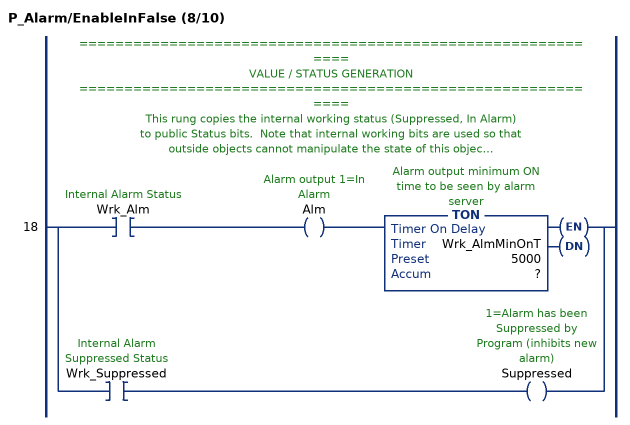
   // ============================================================
   // VALUE / STATUS GENERATION
   // ============================================================
   // This rung copies the internal working status (Suppressed, In Alarm)
   // to public Status bits.  Note that internal working bits are used so that
   // outside objects cannot manipulate the state of this object
   // by setting/clearing its Status and Alarm bits.
   // Public Status is generated for:
   // Alarm (with minimum ON time to be seen by polling)
   // Alarm Suppressed
   // Unsuppressed, Unshelved and Enabled are generated for HMI (FTVSE 7).
   // (Ack, Shelved and Disabled can be set/cleared by the HMI directly.
   // Note that these bits are "read/write" outputs in the parameter definition.)
   // #####  V3.0-00  2013-06-30:  New rung, some from below, new HMI bits.  #####
   18: [XIC(Wrk_Alm) OTE(Alm) TON(Wrk_AlmMinOnT,?,?) ,XIC(Wrk_Suppressed) OTE(Suppressed) ];
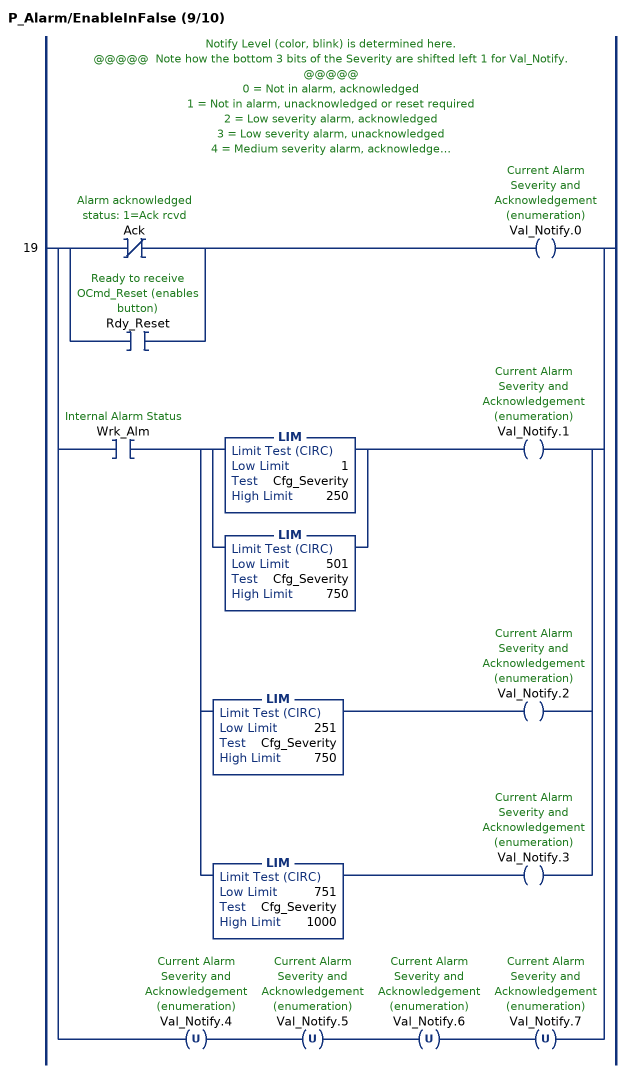
   // Notify Level (color, blink) is determined here.
   // @@@@@  Note how the bottom 3 bits of the Severity are shifted left 1 for Val_Notify.  @@@@@
   // 0 = Not in alarm, acknowledged
   // 1 = Not in alarm, unacknowledged or reset required
   // 2 = Low severity alarm, acknowledged
   // 3 = Low severity alarm, unacknowledged
   // 4 = Medium severity alarm, acknowledged
   // 5 = Medium severity alarm, unacknowledged
   // 6 = High severity alarm, acknowledged
   // 7 = High severity alarm, unacknowledged
   // 8 = Urgent severity alarm, acknowledged
   // 9 = Urgent severity alarm, unacknowledged
   // NOTE that the alarm bell icon will blink, even though the alarm is Acknowledged,
   // if an Alarm Reset is required (to get the Operator's attention).
   // #####  V3.0-00  2013-06-30:  Moved a few functions off this rung to logic above.  #####
   // #####  Names of Severity levels changed to Low, Medium, High, Highest  #####
   // #####  to match examples in ANSI/ISA-18.2-2009.  #####
   // #####  V3.1-00  2014-06-30:  Changed severity ranges, names to match FTAE  #####
   19: [[XIO(Ack) ,XIC(Rdy_Reset) ] OTE(Val_Notify.0) ,XIC(Wrk_Alm) [[LIM(1,Cfg_Severity,250) ,LIM(501,Cfg_Severity,750) ] OTE(Val_Notify.1) ,LIM(251,Cfg_Severity,750) OTE(Val_Notify.2) ,LIM(751,Cfg_Severity,1000) OTE(Val_Notify.3) ] ,OTU(Val_Notify.4) OTU(Val_Notify.5) OTU(Val_Notify.6) OTU(Val_Notify.7) ];
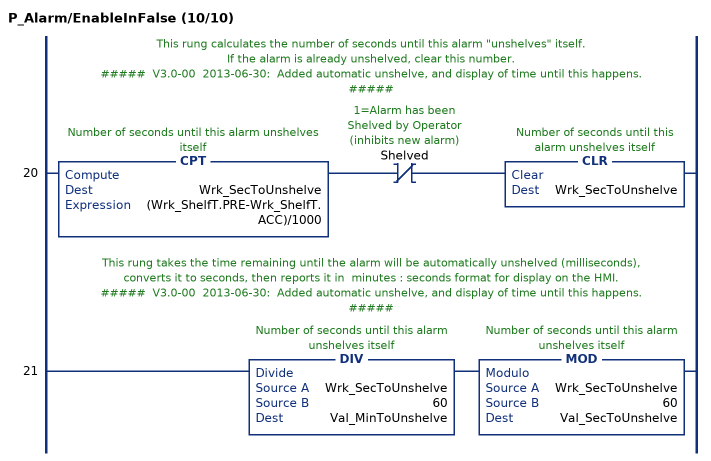
   // This rung calculates the number of seconds until this alarm "unshelves" itself.
   // If the alarm is already unshelved, clear this number.
   // #####  V3.0-00  2013-06-30:  Added automatic unshelve, and display of time until this happens.  #####
   20: CPT(Wrk_SecToUnshelve,(Wrk_ShelfT.PRE-Wrk_ShelfT.ACC)/1000)XIO(Shelved)CLR(Wrk_SecToUnshelve);
   // This rung takes the time remaining until the alarm will be automatically unshelved (milliseconds),
   // converts it to seconds, then reports it in  minutes : seconds format for display on the HMI.
   // #####  V3.0-00  2013-06-30:  Added automatic unshelve, and display of time until this happens.  #####
   21: DIV(Wrk_SecToUnshelve,60,Val_MinToUnshelve)MOD(Wrk_SecToUnshelve,60,Val_SecToUnshelve);
END_ROUTINE
